(* IEC 61131-3 sources: AXOpen/src/core/ctrl/test/AxoMessaging, 3 files *)

(* ---- AxoLogger.st ---- *)
USING AXOpen.Messaging;

NAMESPACE AXOpen.MessagingTests
    {TestFixture}
    CLASS AxoLoggerTest
        VAR
            _sut : AxoLogger;
        END_VAR

        {Test}
        METHOD PUBLIC Log_should_log_info_message
            _sut.Log('this is info message', eLogLevel#Information);
            AxUnit.Assert.Equal(_sut.LogEntries[0].Message, 'this is info message');
            AxUnit.Assert.Equal(true, eLogLevel#Information = _sut.LogEntries[0].Level);
            AxUnit.Assert.Equal(true, _sut.LogEntries[0].ToDequeue);
        END_METHOD

        {Test}
        METHOD PUBLIC MinumuLevel_should_not_set_loggers_min_level
            _sut.MinimumLevel(eLogLevel#Error);
            AxUnit.Assert.Equal(true, eLogLevel#Error = _sut.MinLevel);
        END_METHOD

        // {Test}
        // METHOD PUBLIC Log_should_not_log_message_when_min_level_set_higher
        //     // _sut.MinimumLevel(eLogLevel#Error);
        //     // _sut.Log('this is verbose message', eLogLevel#Verbose);
        //     // AxUnit.Assert.Equal(_sut.LogEntries[0].Message, '');
        //     // AxUnit.Assert.Equal(true, _sut.LogEntries[0].ToDequeue);
        //     // //AxUnit.Assert.Equal(true, eLogLevel#NoCat = _sut.LogEntries[0].Level);
        //     AxUnit.Assert.Equal(TRUE, TRUE);
        // END_METHOD
    END_CLASS
END_NAMESPACE

(* ---- MockAxoContext.st ---- *)
USING AXOpen.Rtc;
USING AXOpen.Messaging;
USING AXOpen.Logging;

NAMESPACE AXOpen.Core
    ///<summary>
    /// Provides base for contextualized entry of `AXOpen` application.
    /// This class is abstract and must be inherited.
    ///</summary>
    {S7.extern=ReadWrite}
    CLASS PUBLIC ABSTRACT MockAxoContext IMPLEMENTS IAxoContext
        VAR PRIVATE
            _openCounter : ULINT;
            _closeCounter : ULINT;
            _identityCounter : ULINT;
            _messagingLevel : eAxoMessageCategory;
         END_VAR

        ///<summary>
        /// The entry point for the context. The call tree of the context start here and all the logic of given context
        /// must be placed here.
        /// This method must be overridden in derived class.
        ///</summary>
        METHOD PROTECTED ABSTRACT Main END_METHOD

        METHOD PRIVATE Open : ULINT
            _openCounter := _openCounter + ULINT#1;
        END_METHOD

        METHOD PRIVATE Close : ULINT
            _closeCounter := _closeCounter + ULINT#1;
        END_METHOD

        ///<summary>
        /// Runs the cycle of this context. This method must be called cyclically in a PLC task.
        ///</summary>
        METHOD PUBLIC Run
            THIS.Open();
            THIS.Main();
            THIS.Close();
        END_METHOD

        ///<summary>
        /// Gets the value of current context cycle counter.
        ///</summary>
        METHOD PUBLIC OpenCycleCount : ULINT
            OpenCycleCount := _openCounter;
        END_METHOD

        METHOD PUBLIC ClosedCycleCount : ULINT
            ClosedCycleCount := _closeCounter;
        END_METHOD

        METHOD PUBLIC CreateIdentity : ULINT
            _identityCounter := _identityCounter + ULINT#1;
            CreateIdentity := _identityCounter;
        END_METHOD

        METHOD PUBLIC PeekIdentity : ULINT
            PeekIdentity := _identityCounter;
        END_METHOD

        VAR PRIVATE
            NULL_RTC : _NULL_RTC;
            _rtc : IAxoRtc;
        END_VAR

        METHOD PUBLIC GetRtc : IAxoRtc
            IF(_rtc <> NULL) THEN
                GetRtc := _rtc;
            ELSE
                GetRtc := NULL_RTC;
            END_IF;
        END_METHOD

        METHOD PUBLIC InjectRtc
            VAR_INPUT
                Rtc : IAxoRtc;
            END_VAR
            _rtc := Rtc;
        END_METHOD

        VAR PRIVATE
            NULL_LOGGER : _NULL_LOGGER;
        END_VAR
        METHOD PUBLIC GetLogger : IAxoLogger GetLogger := NULL_LOGGER; END_METHOD
        METHOD PUBLIC InjectLogger VAR_INPUT _logger : IAxoLogger; END_VAR ; END_METHOD
    END_CLASS
END_NAMESPACE

(* ---- MockAxoObject.st ---- *)
USING AXOpen.Rtc;

NAMESPACE AXOpen.Core
    ///<summary>
    /// Provides base class for all classes of `AXOpen`.
    ///</summary>
    {S7.extern=ReadWrite}
    CLASS PUBLIC MockAxoObject IMPLEMENTS IAxoObject
        VAR PUBLIC
            {#ix-attr:[CompilerOmits("POCO")]}
            {#ix-attr:[ReadOnly()]}
            {#ix-attr:[RenderIgnore()]}
            Identity   : ULINT := ULINT#0;
        END_VAR

        VAR PRIVATE
            _parent     : IAxoObject;
            _context    : IAxoContext;
        END_VAR

        VAR PRIVATE
            {S7.extern=Hidden}
            NULL_CONTEXT : _NULL_CONTEXT;
            {S7.extern=Hidden}
            NULL_OBJECT : _NULL_OBJECT;
        END_VAR

        ///<summary>
        /// Gets unique identity of this object in given context.
        ///</summary>
        METHOD PUBLIC GetIdentity : ULINT
            GetIdentity := Identity;
        END_METHOD

        ///<summary>
        /// Gets context in which this object was initialized.
        ///</summary>
        METHOD PUBLIC GetContext : IAxoContext
            IF(_context <> NULL) THEN
                GetContext := _context;
            ELSE
                GetContext := NULL_CONTEXT;
            END_IF;
        END_METHOD

        METHOD PUBLIC GetContextUnsafe : IAxoContext
                GetContextUnsafe := _context;
        END_METHOD

        ///<summary>
        /// Gets parent in which this object was initialized.
        ///</summary>
        METHOD PUBLIC GetParent : IAxoObject
            IF(_context <> NULL) THEN
                GetParent := _parent;
            ELSE
                GetParent := NULL_OBJECT;
            END_IF;
        END_METHOD

        ///<summary>
        /// Initializes this object associating it given parent.
        /// This method should be called only once upon the program start.
        /// Any subsequent call are ignored.
        ///</summary>
        METHOD PUBLIC Initialize
            VAR_INPUT
                parent : IAxoObject;
            END_VAR

            IF(Identity = ULINT#0 AND parent <> NULL) THEN
                _context    := parent.GetContext();
                Identity   := _context.CreateIdentity();
                _parent     := parent;
                RETURN;
            END_IF;

        END_METHOD

        ///<summary>
        /// Initializes this object associating it given context.
        /// This method should be called only once upon the program start.
        /// Any subsequent call are ignored.
        ///</summary>
        METHOD PUBLIC Initialize
            VAR_INPUT
                context : IAxoContext;
            END_VAR

            IF(Identity = ULINT#0 AND context <> NULL) THEN
                _context    := context;
                Identity   := _context.CreateIdentity();
            END_IF;

        END_METHOD
    END_CLASS
END_NAMESPACE
